TYPE OffsetDistacco :
STRUCT
	Lastra 	: StrutturaGenericaQuotaAssi; 
	Falda 	: StrutturaGenericaQuotaAssi;
END_STRUCT
END_TYPE

(* stored: Version 1.1.0.1, ProductVersion 3.1.4024.11
   DUT OffsetDistacco: Id {6f9cb4cf-9bb7-4a0d-b8ed-ce4d284c2397} *)
